Staubli VAL3: listcreate.pgx

public program listcreate(string x_sTitle)
begin
  //
  // Staubli Copyright 2003 07 31
  //
  sTitle=x_sTitle
  call listframe(sTitle,nTopX,nTopY,nBottomX,nBottomY)
  call listempty()

end
